SYSTEM Test Big Computation par 10
  (* Version 1.0, 2005-12-19, Goran Cengic, Chalmers *)
  DEVICE Test Device : DeviceType_not_used
    RESOURCE Test Resource : ResourceType_not_used
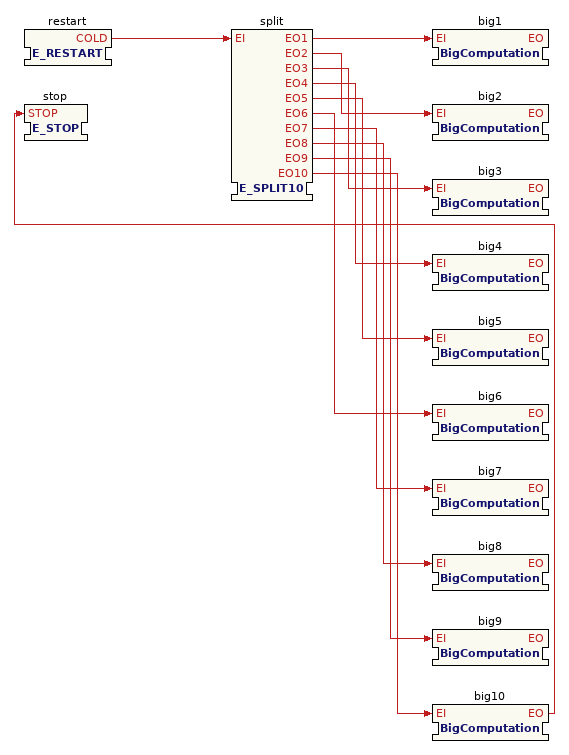
      FBS
        restart : E_RESTART;
        stop : E_STOP;
        split : E_SPLIT10;
        big1 : BigComputation;
        big2 : BigComputation;
        big3 : BigComputation;
        big4 : BigComputation;
        big5 : BigComputation;
        big6 : BigComputation;
        big7 : BigComputation;
        big8 : BigComputation;
        big9 : BigComputation;
        big10 : BigComputation;
      END_FBS
      EVENT_CONNECTIONS
        restart.COLD TO split.EI;
        split.EO1 TO big1.EI;
        split.EO2 TO big2.EI;
        split.EO3 TO big3.EI;
        split.EO4 TO big4.EI;
        split.EO5 TO big5.EI;
        split.EO6 TO big6.EI;
        split.EO7 TO big7.EI;
        split.EO8 TO big8.EI;
        split.EO9 TO big9.EI;
        split.EO10 TO big10.EI;
        big10.EO TO stop.STOP;
      END_CONNECTIONS
    END_RESOURCE
  END_DEVICE
END_SYSTEM
